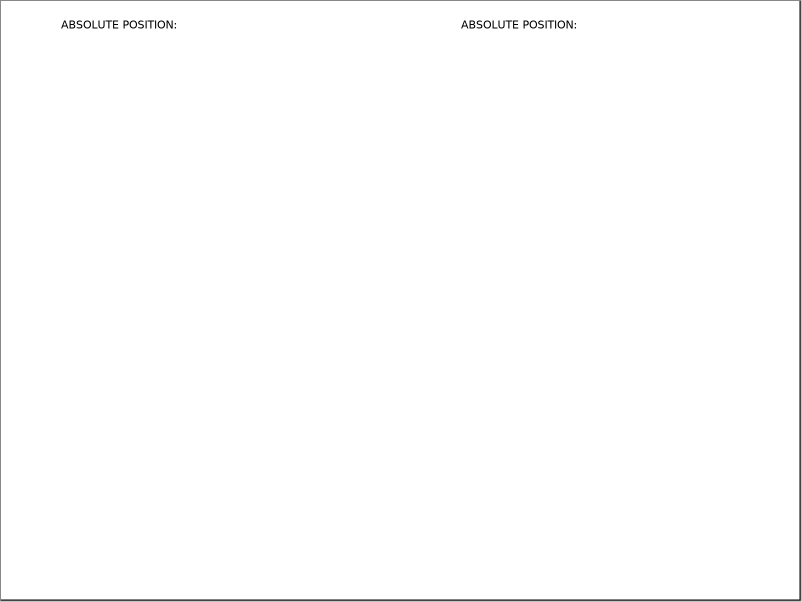
VISUALIZATION F48_Cam_Out  // 802x602
    Rectangle (0,0 800x600)
    Label (10,10 170x30), "ABSOLUTE POSITION:"
    Label (410,10 170x30), "ABSOLUTE POSITION:"
END_VISUALIZATION

(* stored: Version 1.1.0.1, ProductVersion 3.1.4022.7
   Visu F48_Cam_Out: Id {447ec899-ef95-430f-a374-44d967140076} *)
